KUKA KRL data list: Mes_Info_Data.dat

&ACCESS RV
DEFDAT  MES_INFO_DATA PUBLIC

DECL DATE Robot_Run_Time
;GLOBAL ENUM Robot_Process_Name_Enum R_Side_7,R_Side_8,R_Side_9,Panel_Surround_7,Panel_Surround_8,Panel_Surround_9,Panel_Welding_1,Panel_Welding_2,LaserCutting_1,Spot_Surround_1

GLOBAL INT T1_Time=0
GLOBAL INT Aut_Time=0

GLOBAL INT Work_A_Run_Cycle_Time=0
GLOBAL INT Work_A_Run_All_Time=0
GLOBAL INT Work_B_Run_Cycle_Time=0
GLOBAL INT Work_B_Run_All_Time=0
GLOBAL INT Work_C_Run_Cycle_Time=0
GLOBAL INT Work_C_Run_All_Time=0
GLOBAL INT Work_D_Run_Cycle_Time=0
GLOBAL INT Work_D_Run_All_Time=0

GLOBAL BOOL WORK_A_State=FALSE
GLOBAL BOOL WORK_B_State=FALSE
GLOBAL BOOL WORK_C_State=FALSE
GLOBAL BOOL WORK_D_State=FALSE

GLOBAL INT Socket_TimeOut=2000

GLOBAL INT Work_A_Run_Nunber=0
GLOBAL INT Work_B_Run_Nunber=0
GLOBAL INT Work_C_Run_Nunber=0
GLOBAL INT Work_D_Run_Nunber=0
GLOBAL INT Work_All_Run_Nunber=0
GLOBAL CHAR DATAPATH_NAME[1024]



DECL BOOL _Work_A_Stat=FALSE
DECL BOOL _Work_B_Stat=FALSE
DECL BOOL _Work_C_Stat=FALSE
DECL BOOL _Work_D_Stat=FALSE
DECL BOOL _EKRL_Connect_Stat=TRUE
DECL BOOL _EKRL_Send_Stat=TRUE

DECL BOOL _EKRL_Server_Connt_Stat=FALSE

GLOBAL CONST CHAR Robot_Process_Name[1024]
Robot_Process_Name[]="Spot_Sink_8"







ENDDAT
